Fanuc KAREL source: ka00054.KL

-- PROVISIONAL review KL for V940-1; original PC SHA256 58dd9d527f61ae76ee16a5de3c94bdc9cc5275d3f1dbe1fa6dd15e20054318c2
-- Incomplete behavior may be omitted. Consult companion uncertainty JSON. Do not deploy.
PROGRAM KA00054
%NOLOCKGROUP
-- UNRESOLVED_DECL SRC type=000101
-- UNRESOLVED_DECL DST type=000102
BEGIN
  -- V9_ZERO_TABLE_METADATA_HINT layout=0001; no indexed target words; source/name/runtime held
  -- UNRESOLVED_PC offsets 5-25; opcodes 49,7E,4A
  -- UNRESOLVED_PC offsets 30-34; opcodes 7F
END KA00054
